(* Logix 5000 project; controller FRIST_EXAMPLE Emulate 5570 rev 19.11; software revision 19.01 *)

TASK MainTask (continuous, watchdog 500 ms) : MainProgram

MODULES
   Local : Emulate 5570 (ICP 2, rev 19.11)
       : 1756-IB32 (ICP 3, rev 3.1, Input RPI 20 ms)   // DG-INPUT
       : vendor 1 type 7 code 8 (ICP 4, rev 3.1, Output RPI 20 ms)
       : 1756-IF6I (ICP 5, rev 1.1, Input RPI 100 ms)
       : 1756-OF8 (ICP 6, rev 1.1, Output RPI 12 ms)
END_MODULES

VAR_GLOBAL   (* controller tags *)
   CMD_MT01 : BOOL;
   DESLIGA : BOOL := 1;
   LIGA : BOOL;
END_VAR

PROGRAM MainProgram   (* main routine MainRoutine *)
VAR
   CALC : DINT := 7;
   i : DINT;   // iterator
   maior : DINT;
   menor : DINT;
   PARAM1 : DINT := 4;
   PARAM2 : DINT := 3;
   RESULTADO : DINT := 7;
   tabela_busca : DINT[11] := ([0] := 33, [1] := 37, [2] := 255, [3] := 4, [4] := 80, [5] := 457, [6] := 64, [7] := 88, [8] := 92, [9] := 17, [10] := 7);
   VAR1 : DINT := 4;
   VAR2 : DINT := 3;
END_VAR

ROUTINE MainRoutine   (* ladder *)
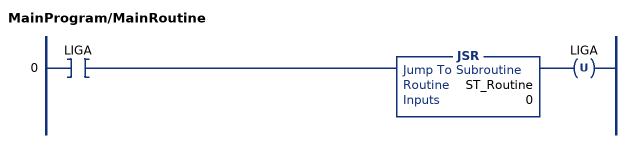
   0: XIC(LIGA)JSR(ST_Routine,0)OTU(LIGA);
END_ROUTINE

ROUTINE ST_Routine   (* structured text *)
   // Retorna maior e menor número
   
   maior := tabela_busca[0];
   menor := tabela_busca[0];
   
   for i:= 0 to 10 by 1
   do
   	if (tabela_busca[i] > maior)
   	then
   		maior := tabela_busca[i];
   	end_if;
   	if (tabela_busca[i] < menor)
   	then
   		menor := tabela_busca[i];
   	end_if;
   end_for;
   
   
   
END_ROUTINE
END_PROGRAM
